   cmJRWinderRearAxisY.commandConfiguration.posRelative.velocity := -1.0;
   cmJRWinderRearAxisY.commandConfiguration.posRelative.acceleration := -1.0;
   cmJRWinderRearAxisY.commandConfiguration.posRelative.deceleration := -1.0;
   cmJRWinderRearAxisY.commandConfiguration.posRelative.jerk := -1.0;
   cmJRWinderRearAxisY.commandConfiguration.posRelative.direction := 0;
   cmJRWinderRearAxisY.commandConfiguration.posAbsolute.position := 0.0;
   cmJRWinderRearAxisY.commandConfiguration.posAbsolute.velocity := -1.0;
   cmJRWinderRearAxisY.commandConfiguration.posAbsolute.acceleration := -1.0;
   cmJRWinderRearAxisY.commandConfiguration.posAbsolute.deceleration := -1.0;
   cmJRWinderRearAxisY.commandConfiguration.posAbsolute.jerk := -1.0;
   cmJRWinderRearAxisY.commandConfiguration.posAbsolute.direction := 1;
   cmJRWinderRearAxisY.commandConfiguration.posAbsolute.positionChangeOnTheFly := FALSE;
   cmJRWinderRearAxisY.commandConfiguration.posAbsolute.velocityChangeOnTheFly := FALSE;
   cmJRWinderRearAxisY.commandConfiguration.posSuperimposed.distance := 0.0;
   cmJRWinderRearAxisY.commandConfiguration.posSuperimposed.velocityDiff := -1.0;
   cmJRWinderRearAxisY.commandConfiguration.posSuperimposed.acceleration := -1.0;
   cmJRWinderRearAxisY.commandConfiguration.posSuperimposed.deceleration := -1.0;
   cmJRWinderRearAxisY.commandConfiguration.posSuperimposed.jerk := -1.0;
   cmJRWinderRearAxisY.commandConfiguration.posSuperimposed.direction := 0;
   cmJRWinderRearAxisY.commandConfiguration.haltSuperimposed.deceleration := -1.0;
   cmJRWinderRearAxisY.commandConfiguration.haltSuperimposed.jerk := -1.0;
   cmJRWinderRearAxisY.commandConfiguration.haltSuperimposed.abortAcceleration := FALSE;
   cmJRWinderRearAxisY.commandConfiguration.gearInRelative.ratioNumerator := 1;
   cmJRWinderRearAxisY.commandConfiguration.gearInRelative.ratioDenominator := 1;
   cmJRWinderRearAxisY.commandConfiguration.gearInRelative.acceleration := -1.0;
   cmJRWinderRearAxisY.commandConfiguration.gearInRelative.deceleration := -1.0;
   cmJRWinderRearAxisY.commandConfiguration.gearInRelative.jerk := -1.0;
   cmJRWinderRearAxisY.commandConfiguration.gearInRelative.ratioChangeOnTheFly := FALSE;
   cmJRWinderRearAxisY.commandConfiguration.gearInAbsolute.ratioNumerator := 1;
   cmJRWinderRearAxisY.commandConfiguration.gearInAbsolute.ratioDenominator := 1;
   cmJRWinderRearAxisY.commandConfiguration.gearInAbsolute.masterSyncPosition := 0.0;
   cmJRWinderRearAxisY.commandConfiguration.gearInAbsolute.slaveSyncPosition := 0.0;
   cmJRWinderRearAxisY.commandConfiguration.gearInAbsolute.syncProfileReference := 1;
   cmJRWinderRearAxisY.commandConfiguration.gearInAbsolute.masterStartDistance := 0.0;
   cmJRWinderRearAxisY.commandConfiguration.gearInAbsolute.velocity := -1.0;
   cmJRWinderRearAxisY.commandConfiguration.gearInAbsolute.acceleration := -1.0;
   cmJRWinderRearAxisY.commandConfiguration.gearInAbsolute.deceleration := -1.0;
   cmJRWinderRearAxisY.commandConfiguration.gearInAbsolute.jerk := -1.0;
   cmJRWinderRearAxisY.commandConfiguration.gearInAbsolute.syncDirection := 1;
   cmJRWinderRearAxisY.commandConfiguration.gearInAbsolute.ratioChangeOnTheFly := FALSE;
   cmJRWinderRearAxisY.commandConfiguration.gearInVelocity.continuousUpdate := FALSE;
   cmJRWinderRearAxisY.commandConfiguration.gearInVelocity.ratioNumerator := 1;
   cmJRWinderRearAxisY.commandConfiguration.gearInVelocity.ratioDenominator := 1;
   cmJRWinderRearAxisY.commandConfiguration.gearInVelocity.acceleration := -1.0;
   cmJRWinderRearAxisY.commandConfiguration.gearInVelocity.deceleration := -1.0;
   cmJRWinderRearAxisY.commandConfiguration.gearInVelocity.jerk := -1.0;
   cmJRWinderRearAxisY.commandConfiguration.gearInVelocity.positionControlled := FALSE;
   cmJRWinderRearAxisY.commandConfiguration.camIn.masterOffset := 0.0;
   cmJRWinderRearAxisY.commandConfiguration.camIn.slaveOffset := 0.0;
   cmJRWinderRearAxisY.commandConfiguration.camIn.masterScaling := 1.0;
   cmJRWinderRearAxisY.commandConfiguration.camIn.slaveScaling := 1.0;
   cmJRWinderRearAxisY.commandConfiguration.camIn.masterSyncPosition := 0.0;
   cmJRWinderRearAxisY.commandConfiguration.camIn.syncProfileReference := 1;
   cmJRWinderRearAxisY.commandConfiguration.camIn.masterStartDistance := 0.0;
   cmJRWinderRearAxisY.commandConfiguration.camIn.velocity := -1.0;
   cmJRWinderRearAxisY.commandConfiguration.camIn.acceleration := -1.0;
   cmJRWinderRearAxisY.commandConfiguration.camIn.deceleration := -1.0;
   cmJRWinderRearAxisY.commandConfiguration.camIn.jerk := -1.0;
   cmJRWinderRearAxisY.commandConfiguration.camIn.applicationMode := 0;
   cmJRWinderRearAxisY.commandConfiguration.camIn.syncDirection := 1;
   cmJRWinderRearAxisY.commandConfiguration.gearOutCamOut.slavePosition := 0.0;
   cmJRWinderRearAxisY.commandConfiguration.gearOutCamOut.syncProfileReference := 1;
   cmJRWinderRearAxisY.commandConfiguration.gearOutCamOut.masterStopDistance := 0.0;
   cmJRWinderRearAxisY.commandConfiguration.gearOutCamOut.deceleration := -1.0;
   cmJRWinderRearAxisY.commandConfiguration.gearOutCamOut.jerk := -1.0;
   cmJRWinderRearAxisY.commandConfiguration.gearOutCamOut.syncOutDirection := 3;
   cmJRWinderRearAxisY.commandConfiguration.gearOutCamOut.gearOutCamOutMode := -1;
   cmJRWinderRearAxisY.commandConfiguration.phasing.phaseShift := 0.0;
   cmJRWinderRearAxisY.commandConfiguration.phasing.velocity := -1.0;
   cmJRWinderRearAxisY.commandConfiguration.phasing.acceleration := -1.0;
   cmJRWinderRearAxisY.commandConfiguration.phasing.deceleration := -1.0;
   cmJRWinderRearAxisY.commandConfiguration.phasing.jerk := -1.0;
   cmJRWinderRearAxisY.commandConfiguration.phasing.profileReference := 0;
   cmJRWinderRearAxisY.commandConfiguration.phasing.phasingDistance := 0.0;
   cmJRWinderRearAxisY.commandConfiguration.phasing.startPosition := 0.0;
   cmJRWinderRearAxisY.commandConfiguration.phasing.direction := 3;
   cmJRWinderRearAxisY.commandConfiguration.phasing.phaseAbsolute := TRUE;
   cmJRWinderRearAxisY.commandConfiguration.phasing.phaseShiftChangeOnTheFly := FALSE;
   cmJRWinderRearAxisY.commandConfiguration.offset.offset := 0.0;
   cmJRWinderRearAxisY.commandConfiguration.offset.profileReference := 1;
   cmJRWinderRearAxisY.commandConfiguration.offset.offsetDistance := 0.0;
   cmJRWinderRearAxisY.commandConfiguration.offset.startPosition := 0.0;
   cmJRWinderRearAxisY.commandConfiguration.offset.direction := 3;
   cmJRWinderRearAxisY.commandConfiguration.offset.offsetAbsolute := TRUE;
   cmJRWinderRearAxisY.commandConfiguration.offset.offsetChangeOnTheFly := FALSE;
   cmJRWinderRearAxisY.monitoring.valid := FALSE;
   cmJRWinderRearAxisY.monitoring.busy := TRUE;
   cmJRWinderRearAxisY.monitoring.error := TRUE;
   cmJRWinderRearAxisY.monitoring.status := 16#8600;
   cmJRWinderRearAxisY.monitoring.subfunctionStatus := 16#8001;
   cmJRWinderRearAxisY.monitoring.axisEnabled := FALSE;
   cmJRWinderRearAxisY.monitoring.resetActive := FALSE;
   cmJRWinderRearAxisY.monitoring.inVelocity := FALSE;
   cmJRWinderRearAxisY.monitoring.inLimitation := FALSE;
   cmJRWinderRearAxisY.monitoring.inClamping := FALSE;
   cmJRWinderRearAxisY.monitoring.startSync := FALSE;
   cmJRWinderRearAxisY.monitoring.inSync := FALSE;
   cmJRWinderRearAxisY.monitoring.inSimulation := FALSE;
   cmJRWinderRearAxisY.monitoring.jogSelected := FALSE;
   cmJRWinderRearAxisY.monitoring.moveVelocitySelected := FALSE;
   cmJRWinderRearAxisY.monitoring.stopSelected := FALSE;
   cmJRWinderRearAxisY.monitoring.fastStopSelected := FALSE;
   cmJRWinderRearAxisY.monitoring.torqueLimitingSelected := FALSE;
   cmJRWinderRearAxisY.monitoring.homingSelected := FALSE;
   cmJRWinderRearAxisY.monitoring.posRelativeSelected := FALSE;
   cmJRWinderRearAxisY.monitoring.posAbsoluteSelected := FALSE;
   cmJRWinderRearAxisY.monitoring.posSuperimposedSelected := FALSE;
   cmJRWinderRearAxisY.monitoring.haltSuperimposedSelected := FALSE;
   cmJRWinderRearAxisY.monitoring.commandBusy := FALSE;
   cmJRWinderRearAxisY.monitoring.commandDone := FALSE;
   cmJRWinderRearAxisY.monitoring.commandAborted := FALSE;
   cmJRWinderRearAxisY.monitoring.homingCommandBusy := FALSE;
   cmJRWinderRearAxisY.monitoring.homingCommandDone := FALSE;
   cmJRWinderRearAxisY.monitoring.homingCommandAborted := FALSE;
   cmJRWinderRearAxisY.monitoring.superimposedBusy := FALSE;
   cmJRWinderRearAxisY.monitoring.superimposedDone := FALSE;
   cmJRWinderRearAxisY.monitoring.superimposedAborted := FALSE;
   cmJRWinderRearAxisY.monitoring.actualPosition := -17.994;
   cmJRWinderRearAxisY.monitoring.actualSpeed := 0.0;
   cmJRWinderRearAxisY.monitoring.speedUnit := 1062;
   cmJRWinderRearAxisY.monitoring.positionUnit := 1013;
   cmJRWinderRearAxisY.monitoring.axisType := 1;
   cmJRWinderRearAxisY.monitoring.interlockGeneralOut := TRUE;
   cmJRWinderRearAxisY.monitoring.interlockJogForwardOut := TRUE;
   cmJRWinderRearAxisY.monitoring.interlockJogBackwardOut := TRUE;
   cmJRWinderFrontAxisY.commandConfiguration.power.startMode := 1;
   cmJRWinderFrontAxisY.commandConfiguration.power.stopMode := 0;
   cmJRWinderFrontAxisY.commandConfiguration.power.syncMotionSimulation := FALSE;
   cmJRWinderFrontAxisY.commandConfiguration.power.syncMotionSimulationExtendedMode := -1;
   cmJRWinderFrontAxisY.commandConfiguration.jog.velocity := 0.0;
   cmJRWinderFrontAxisY.commandConfiguration.jog.acceleration := -1.0;
   cmJRWinderFrontAxisY.commandConfiguration.jog.deceleration := -1.0;
   cmJRWinderFrontAxisY.commandConfiguration.jog.jerk := -1.0;
   cmJRWinderFrontAxisY.commandConfiguration.jog.positionControlled := TRUE;
   cmJRWinderFrontAxisY.commandConfiguration.jog.increment := 0.0;
   cmJRWinderFrontAxisY.commandConfiguration.jog.mode := 0;
   cmJRWinderFrontAxisY.commandConfiguration.moveVelocity.velocity := 0.0;
   cmJRWinderFrontAxisY.commandConfiguration.moveVelocity.acceleration := -1.0;
   cmJRWinderFrontAxisY.commandConfiguration.moveVelocity.deceleration := -1.0;
   cmJRWinderFrontAxisY.commandConfiguration.moveVelocity.jerk := -1.0;
   cmJRWinderFrontAxisY.commandConfiguration.moveVelocity.direction := 0;
   cmJRWinderFrontAxisY.commandConfiguration.moveVelocity.positionControlled := TRUE;
   cmJRWinderFrontAxisY.commandConfiguration.moveVelocity.velocityChangeOnTheFly := FALSE;
   cmJRWinderFrontAxisY.commandConfiguration.stop.deceleration := -1.0;
   cmJRWinderFrontAxisY.commandConfiguration.stop.jerk := -1.0;
   cmJRWinderFrontAxisY.commandConfiguration.stop.abortAcceleration := FALSE;
   cmJRWinderFrontAxisY.commandConfiguration.fastStop.deceleration := -1.0;
   cmJRWinderFrontAxisY.commandConfiguration.fastStop.jerk := -1.0;
   cmJRWinderFrontAxisY.commandConfiguration.fastStop.abortAcceleration := FALSE;
   cmJRWinderFrontAxisY.commandConfiguration.fastStop.replaceStopPossible := FALSE;
   cmJRWinderFrontAxisY.commandConfiguration.torqueLimiting.limit := -1.0;
   cmJRWinderFrontAxisY.commandConfiguration.torqueLimiting.mode := 0;
   cmJRWinderFrontAxisY.commandConfiguration.homing.position := 0.0;
   cmJRWinderFrontAxisY.commandConfiguration.homing.mode := 0;
   cmJRWinderFrontAxisY.commandConfiguration.homing.sensor := 0;
   cmJRWinderFrontAxisY.commandConfiguration.homing.extendedMode := -1;
   cmJRWinderFrontAxisY.commandConfiguration.homing.extendedModeTorqueLimit := 0.0;
   cmJRWinderFrontAxisY.commandConfiguration.homing.extendedModeTargetPosition := 0.0;
   cmJRWinderFrontAxisY.commandConfiguration.posRelative.distance := 0.0;
   cmJRWinderFrontAxisY.commandConfiguration.posRelative.velocity := -1.0;
   cmJRWinderFrontAxisY.commandConfiguration.posRelative.acceleration := -1.0;
   cmJRWinderFrontAxisY.commandConfiguration.posRelative.deceleration := -1.0;
   cmJRWinderFrontAxisY.commandConfiguration.posRelative.jerk := -1.0;
   cmJRWinderFrontAxisY.commandConfiguration.posRelative.direction := 0;
   cmJRWinderFrontAxisY.commandConfiguration.posAbsolute.position := 0.0;
   cmJRWinderFrontAxisY.commandConfiguration.posAbsolute.velocity := -1.0;
   cmJRWinderFrontAxisY.commandConfiguration.posAbsolute.acceleration := -1.0;
   cmJRWinderFrontAxisY.commandConfiguration.posAbsolute.deceleration := -1.0;
   cmJRWinderFrontAxisY.commandConfiguration.posAbsolute.jerk := -1.0;
   cmJRWinderFrontAxisY.commandConfiguration.posAbsolute.direction := 1;
   cmJRWinderFrontAxisY.commandConfiguration.posAbsolute.positionChangeOnTheFly := FALSE;
   cmJRWinderFrontAxisY.commandConfiguration.posAbsolute.velocityChangeOnTheFly := FALSE;
   cmJRWinderFrontAxisY.commandConfiguration.posSuperimposed.distance := 0.0;
   cmJRWinderFrontAxisY.commandConfiguration.posSuperimposed.velocityDiff := -1.0;
   cmJRWinderFrontAxisY.commandConfiguration.posSuperimposed.acceleration := -1.0;
   cmJRWinderFrontAxisY.commandConfiguration.posSuperimposed.deceleration := -1.0;
   cmJRWinderFrontAxisY.commandConfiguration.posSuperimposed.jerk := -1.0;
   cmJRWinderFrontAxisY.commandConfiguration.posSuperimposed.direction := 0;
   cmJRWinderFrontAxisY.commandConfiguration.haltSuperimposed.deceleration := -1.0;
   cmJRWinderFrontAxisY.commandConfiguration.haltSuperimposed.jerk := -1.0;
   cmJRWinderFrontAxisY.commandConfiguration.haltSuperimposed.abortAcceleration := FALSE;
   cmJRWinderFrontAxisY.commandConfiguration.gearInRelative.ratioNumerator := 1;
   cmJRWinderFrontAxisY.commandConfiguration.gearInRelative.ratioDenominator := 1;
   cmJRWinderFrontAxisY.commandConfiguration.gearInRelative.acceleration := -1.0;
   cmJRWinderFrontAxisY.commandConfiguration.gearInRelative.deceleration := -1.0;
   cmJRWinderFrontAxisY.commandConfiguration.gearInRelative.jerk := -1.0;
   cmJRWinderFrontAxisY.commandConfiguration.gearInRelative.ratioChangeOnTheFly := FALSE;
   cmJRWinderFrontAxisY.commandConfiguration.gearInAbsolute.ratioNumerator := 1;
   cmJRWinderFrontAxisY.commandConfiguration.gearInAbsolute.ratioDenominator := 1;
   cmJRWinderFrontAxisY.commandConfiguration.gearInAbsolute.masterSyncPosition := 0.0;
   cmJRWinderFrontAxisY.commandConfiguration.gearInAbsolute.slaveSyncPosition := 0.0;
   cmJRWinderFrontAxisY.commandConfiguration.gearInAbsolute.syncProfileReference := 1;
   cmJRWinderFrontAxisY.commandConfiguration.gearInAbsolute.masterStartDistance := 0.0;
   cmJRWinderFrontAxisY.commandConfiguration.gearInAbsolute.velocity := -1.0;
   cmJRWinderFrontAxisY.commandConfiguration.gearInAbsolute.acceleration := -1.0;
   cmJRWinderFrontAxisY.commandConfiguration.gearInAbsolute.deceleration := -1.0;
   cmJRWinderFrontAxisY.commandConfiguration.gearInAbsolute.jerk := -1.0;
   cmJRWinderFrontAxisY.commandConfiguration.gearInAbsolute.syncDirection := 1;
   cmJRWinderFrontAxisY.commandConfiguration.gearInAbsolute.ratioChangeOnTheFly := FALSE;
   cmJRWinderFrontAxisY.commandConfiguration.gearInVelocity.continuousUpdate := FALSE;
   cmJRWinderFrontAxisY.commandConfiguration.gearInVelocity.ratioNumerator := 1;
   cmJRWinderFrontAxisY.commandConfiguration.gearInVelocity.ratioDenominator := 1;
   cmJRWinderFrontAxisY.commandConfiguration.gearInVelocity.acceleration := -1.0;
   cmJRWinderFrontAxisY.commandConfiguration.gearInVelocity.deceleration := -1.0;
   cmJRWinderFrontAxisY.commandConfiguration.gearInVelocity.jerk := -1.0;
   cmJRWinderFrontAxisY.commandConfiguration.gearInVelocity.positionControlled := FALSE;
   cmJRWinderFrontAxisY.commandConfiguration.camIn.masterOffset := 0.0;
   cmJRWinderFrontAxisY.commandConfiguration.camIn.slaveOffset := 0.0;
   cmJRWinderFrontAxisY.commandConfiguration.camIn.masterScaling := 1.0;
   cmJRWinderFrontAxisY.commandConfiguration.camIn.slaveScaling := 1.0;
   cmJRWinderFrontAxisY.commandConfiguration.camIn.masterSyncPosition := 0.0;
   cmJRWinderFrontAxisY.commandConfiguration.camIn.syncProfileReference := 1;
   cmJRWinderFrontAxisY.commandConfiguration.camIn.masterStartDistance := 0.0;
   cmJRWinderFrontAxisY.commandConfiguration.camIn.velocity := -1.0;
   cmJRWinderFrontAxisY.commandConfiguration.camIn.acceleration := -1.0;
   cmJRWinderFrontAxisY.commandConfiguration.camIn.deceleration := -1.0;
   cmJRWinderFrontAxisY.commandConfiguration.camIn.jerk := -1.0;
   cmJRWinderFrontAxisY.commandConfiguration.camIn.applicationMode := 0;
   cmJRWinderFrontAxisY.commandConfiguration.camIn.syncDirection := 1;
   cmJRWinderFrontAxisY.commandConfiguration.gearOutCamOut.slavePosition := 0.0;
   cmJRWinderFrontAxisY.commandConfiguration.gearOutCamOut.syncProfileReference := 1;
   cmJRWinderFrontAxisY.commandConfiguration.gearOutCamOut.masterStopDistance := 0.0;
   cmJRWinderFrontAxisY.commandConfiguration.gearOutCamOut.deceleration := -1.0;
   cmJRWinderFrontAxisY.commandConfiguration.gearOutCamOut.jerk := -1.0;
   cmJRWinderFrontAxisY.commandConfiguration.gearOutCamOut.syncOutDirection := 3;
   cmJRWinderFrontAxisY.commandConfiguration.gearOutCamOut.gearOutCamOutMode := -1;
   cmJRWinderFrontAxisY.commandConfiguration.phasing.phaseShift := 0.0;
   cmJRWinderFrontAxisY.commandConfiguration.phasing.velocity := -1.0;
   cmJRWinderFrontAxisY.commandConfiguration.phasing.acceleration := -1.0;
   cmJRWinderFrontAxisY.commandConfiguration.phasing.deceleration := -1.0;
   cmJRWinderFrontAxisY.commandConfiguration.phasing.jerk := -1.0;
   cmJRWinderFrontAxisY.commandConfiguration.phasing.profileReference := 0;
   cmJRWinderFrontAxisY.commandConfiguration.phasing.phasingDistance := 0.0;
   cmJRWinderFrontAxisY.commandConfiguration.phasing.startPosition := 0.0;
   cmJRWinderFrontAxisY.commandConfiguration.phasing.direction := 3;
   cmJRWinderFrontAxisY.commandConfiguration.phasing.phaseAbsolute := TRUE;
   cmJRWinderFrontAxisY.commandConfiguration.phasing.phaseShiftChangeOnTheFly := FALSE;
   cmJRWinderFrontAxisY.commandConfiguration.offset.offset := 0.0;
   cmJRWinderFrontAxisY.commandConfiguration.offset.profileReference := 1;
   cmJRWinderFrontAxisY.commandConfiguration.offset.offsetDistance := 0.0;
   cmJRWinderFrontAxisY.commandConfiguration.offset.startPosition := 0.0;
   cmJRWinderFrontAxisY.commandConfiguration.offset.direction := 3;
   cmJRWinderFrontAxisY.commandConfiguration.offset.offsetAbsolute := TRUE;
   cmJRWinderFrontAxisY.commandConfiguration.offset.offsetChangeOnTheFly := FALSE;
END_DATA_BLOCK
